(* CODESYS project SingleElevator.project

Project tree, tasks and I/O mapping:
  Device : CODESYS Control Win V3, 3S - Smart Software Solutions GmbH, version 3.5.15.10
    application Application
      libraries: Standard, * (System)
      task MainTask (cyclic, interval 50 ms, priority 1) calls Simulation, GAInstances, Policy
      task VISU_TASK (cyclic, interval 100 ms, priority 31) calls VisuElems.Visu_Prg
      global variables GVL
      visualisation Visualization
      program Simulation [ST]
      function block Motor [SFC]: Closing_active, Closing_exit, Descent_exit, Ascent_active, Ascent_exit, InitFinished_active, Reset_DONEinit_active, Descent_active, Init_active, Ascent_1_active, Descent_1_active, Ready_active, Busy_active, FIN_active, Reset_DONE_active, Ascent_1_exit, CounterUp_active, CounterDown_active, MotStopUp_exit, MotStopDown_exit, Descent_1_exit, Ready_2_active, Busy_2_active, LowSpeed_exit, LowSpeed2_exit, GenCounter_active, ErrDet_active, FaultDeck7_active, Sensor_Fault_active, Error_Floor7_exit, Floor7_active, FloorG_active, AvailableFloor_active, AvailableFloor_exit, FaultDeckG_active, Availablefloor1_active, Availablefloor1_exit
      function block Door [SFC]: Opening_Act_active, Opening_Act_exit, Closing_Act_active, Control_active, Closing_Act_exit, Busy_active, Ready_active, Step1_active, Step1_exit, Init_active, Finished_active, ResetDone_active, Presence_active, Presence_exit, Step3_Closing_Act_active_active, ReOpen_active, ReOpen_exit, Dummy3_exit, ReOpen2_active, ReOpen2_exit
      program Policy [SFC]: Closing_active, Closing_exit, Opening_active, Opening_exit, Motor_Init_exit, Closing_1_active, Closing_1_exit, Upward_active, Upward_exit, Downward_active, Opening_1_active, Opening_1_exit, FloorDetect_active, Motor_Init_active, Downward_exit, ERROR_ARREST_active
      program GAInstances [FBD]
      function block Led [SFC]: GroundFloor_active, Init_active, FirstFloor_active, SecondFloor_active, ThirdFloor_active, FourthFloor_active, FifthFloor_active, SixthFloor_active, SeventhFloor_active, Emergency_active, Ordering_active, Ready_active, Busy_active, Reset_active
  text list GlobalTextList
*)

// Device/Application/GVL
{attribute 'qualified_only'}
VAR_GLOBAL
(* Elevator managing variables*)
	DoorGA_1  	:	Door ;
	MotorGA_1	:	Motor ;
	LedGA_1		:	Led ;

	Open: BOOL;				(* Sensor: the door is fully open*)
	Closed: BOOL;			(* Sensor: the door is fully closed*)
	LimitDown: BOOL;		(* Sensor: lower limit sensor, if TRUE the lift has reached the lower limit*)
	LimitUp: BOOL;			(* Sensor: upper limit sensor, if TRUE the lift has reached the upper limit*)
	DeckSensor: BOOL;		(* Sensor: if TRUE the cab is in proximity of a deck*)
	RampSensor: BOOL;		(* Sensor: if TRUE the cab is in proximity of a ramp*)
	Presence :BOOL; 		(* Sensor: if TRUE something blocks the door photocell*)
	Emergency: BOOL;		(* Input: if TRUE the emergency button has been pressed*)

	Closing: BOOL;			(* Actuator: if TRUE the door starts closing*)
	Opening: BOOL;			(* Actuator: the door starts opening*)
	Motor_on: BOOL;			(* Actuator: if TRUE the lift pulley motor start moving*)
	Up: BOOL;				(* Actuator parameter: if TRUE the lift moves upward, downward otherwise*)
	Vel: BOOL;				(* Actuator parameter: motor speed, if TRUE high speed, low speed otherwise*)


	Current: INT;  			(* Visualization: variable used to storage the current deck*)
    Destination: INT;		(* Visualization: variable used to storage the the destination deck*)
	EmergencyVis: BOOL; 	(* Visualization: if TRUE the emergency light is turned on*)

	InitialDeck: INT := 1;	(* Only for simulation: variable used to define the initial deck*)
	InitCycle: BOOL := FALSE;(* Only for simulation: used to execute the instruction at the first cycle*)
	Height: INT;			(* Only for simulation: elevator height*)
	DeckRest: INT;        	(* Only for simulation: division rest for generating deck sensor*)
	Memory: INT;
	RampRest: INT;			(* Only for simulation: division rest for generating the ramp position*)
	MemoryR: INT;
	Door: INT;				(* Only for simulation: to visualize the closing of the door*)
	Displacement: INT;		(* Only for simulation: lift displacement, dependent on the motor speed*)
	

 (*Inputs: internal panel variables*)
	PG: BOOL;
	P1: BOOL;
	P2: BOOL;
	P3: BOOL;
	P4: BOOL;
	P5: BOOL;
	P6: BOOL;
	P7: BOOL;

(*Visualization: internal panel variables used to turn on the LED*)
	PGVis: BOOL;
	P1Vis: BOOL;
	P2Vis: BOOL;
	P3Vis: BOOL;
	P4Vis: BOOL;
	P5Vis: BOOL;
	P6Vis: BOOL;
	P7Vis: BOOL;

(*Inputs: external panel variables*)
	UpDeckG: BOOL;
	UpDeck1: BOOL;
	UpDeck2: BOOL;
	UpDeck3: BOOL;
	UpDeck4: BOOL;
	UpDeck5: BOOL;
	UpDeck6: BOOL;
	DownDeck7: BOOL;
	DownDeck6: BOOL;
	DownDeck5: BOOL;
	DownDeck4: BOOL;
	DownDeck3: BOOL;
	DownDeck2: BOOL;
	DownDeck1: BOOL;

(*Visualization: external panel variables used to turn on the LED*)
	UpDeckGVis: BOOL;
	UpDeck1Vis: BOOL;
	UpDeck2Vis: BOOL;
	UpDeck3Vis: BOOL;
	UpDeck4Vis: BOOL;
	UpDeck5Vis: BOOL;
	UpDeck6Vis: BOOL;
	DownDeck7Vis: BOOL;
	DownDeck6Vis: BOOL;
	DownDeck5Vis: BOOL;
	DownDeck4Vis: BOOL;
	DownDeck3Vis: BOOL;
	DownDeck2Vis: BOOL;
	DownDeck1Vis: BOOL;

(*Only for simulation: variables used to simulate the fault on deck sensor*)
	SensorG: BOOL;				(* if TRUE the magnetic information for deck G is lost and the deck sensor cannot become TRUE*)
	Sensor1: BOOL;				(* if TRUE the magnetic information for deck 1 is lost and the deck sensor cannot become TRUE*)
	Sensor2: BOOL;
	Sensor3: BOOL;
	Sensor4: BOOL;
	Sensor5: BOOL;
	Sensor6: BOOL;
	Sensor7: BOOL;
	FaultSensorAlarm: BOOL; 	(* Visulaization: if TRUE alerts the user of a deck sensor fault*)

(*Only for simulation: variables used to simulate the fault on ramp sensor*)
	RampGUp: BOOL;
	Ramp1Down: BOOL;
	Ramp1Up:BOOL;
	Ramp2Down: BOOL;
	Ramp2Up:BOOL;
	Ramp3Down: BOOL;
	Ramp3Up:BOOL;
	Ramp4Down: BOOL;
	Ramp4Up:BOOL;
	Ramp5Down: BOOL;
	Ramp5Up:BOOL;
	Ramp6Down: BOOL;
	Ramp6Up:BOOL;
	Ramp7Down: BOOL;
	FaultRampAlarm: BOOL; 		(* Visulaization: if TRUE alerts the user of a ramp sensor fault*)
	SensorGOK: BOOL;
	Sensor1OK: BOOL;
	Sensor2OK: BOOL;
	Sensor6OK: BOOL;
	Sensor3OK: BOOL;
	Sensor4OK: BOOL;
	Sensor5OK: BOOL;
	Sensor7OK: BOOL;
	RampGUpOK: BOOL;
	Ramp1DownOK: BOOL;
	Ramp1UpOK: BOOL;
	Ramp2DownOK: BOOL;
	Ramp2UpOK: BOOL;
	Ramp3DownOK: BOOL;
	Ramp3UpOK: BOOL;
	Ramp4DownOK: BOOL;
	Ramp4UpOK: BOOL;
	Ramp5DownOK: BOOL;
	Ramp5UpOK: BOOL;
	Ramp6DownOK: BOOL;
	Ramp6UpOK: BOOL;
	Ramp7DownOK: BOOL;
	Ramp7UpOK: BOOL;
END_VAR

// Device/Application/Simulation
PROGRAM Simulation
VAR
END_VAR

(* Initial position of the cab inside the hoistway. It is executed only at the first cycle.  *)
IF NOT GVL.InitCycle THEN
			GVL.InitCycle := TRUE ;
			GVL.Height := 20 * GVL.InitialDeck;
		    GVL.Door := 0;
			GVL.Current := GVL.Height / 20;
END_IF;

(* Elevator management, these instructions are executed each cycle time*)

(* Elevator door control. *)
IF GVL.Closing THEN
	GVL.Door := GVL.Door + 1;		(*Closing door management*)
	GVL.Open := FALSE;
END_IF

IF GVL.Door >= 60 THEN						(* Closed door limit*)
	GVL.Closed := TRUE;
END_IF

IF GVL.Opening THEN
	GVL.Door := GVL.Door - 1; 	(* Opening door management*)
	GVL.Closed := FALSE;
END_IF

IF GVL.Door <= 0 THEN							(* Open door limit*)
	GVL.Open := TRUE;
END_IF


(* Maximum and minimum management in the door simulation*)
IF GVL.Door < 0 THEN
	 GVL.Door := 0;
END_IF

IF GVL.Door > 60 THEN
	GVL.Door := 60;
END_IF


(* Control of the cab position inside the hostway. *)
(* Displacement definition for graphic visualization*)
IF GVL.Vel THEN 
	GVL.Displacement := 2;
ELSE 
	GVL.Displacement := 1;
END_IF


(* Height modification relying on direction and speed*)
IF GVL.Motor_on AND GVL.Up THEN
	GVL.Height := GVL.Height + GVL.Displacement;
	GVL.LimitDown := FALSE;
END_IF

IF GVL.Motor_on AND NOT GVL.Up THEN
	GVL.Height := GVL.Height - GVL.Displacement;
	GVL.LimitUp := FALSE;
END_IF


(* Limits for visualization*)
IF GVL.Height < -20 THEN
	GVL.Height := -20;
END_IF

IF GVL.Height > 160 THEN
	GVL.Height := 160;
END_IF

(* Limit sensors management*)
IF GVL.Height <= -10 THEN
	GVL.LimitDown := TRUE;
END_IF

IF GVL.Height >= 150 THEN
	 GVL.LimitUp := TRUE;
END_IF


(*-------------------------------------------------------------------*)
(*  Fault Management (Deck and Ramp Sensors)   *)
(*-------------------------------------------------------------------*)
(* Deck Sensor*)
(* Range of value where the deck sensor is active*)
IF ((GVL.Height >= -1) AND (GVL.Height <= 1)) THEN
	GVL.SensorGOK := TRUE;
ELSE  
	GVL.SensorGOK := FALSE;
END_IF

IF ((GVL.Height >= 20-1) AND (GVL.Height <= 20+1)) THEN
	GVL.Sensor1OK := TRUE;
ELSE  
	GVL.Sensor1OK := FALSE;
END_IF

IF ((GVL.Height >= 40-1) AND (GVL.Height <= 40+1)) THEN
	GVL.Sensor2OK := TRUE;
ELSE  
	GVL.Sensor2OK := FALSE;
END_IF

IF ((GVL.Height >= 60-1) AND (GVL.Height <= 60+1)) THEN
	GVL.Sensor3OK := TRUE;
ELSE  
	GVL.Sensor3OK := FALSE;
END_IF

IF ((GVL.Height >= 80-1) AND (GVL.Height <= 80+1)) THEN
	GVL.Sensor4OK := TRUE;
ELSE  
	GVL.Sensor4OK := FALSE;
END_IF

IF ((GVL.Height >= 100-1) AND (GVL.Height <= 100+1)) THEN
	GVL.Sensor5OK := TRUE;
ELSE   
	GVL.Sensor5OK := FALSE;
END_IF

IF ((GVL.Height >= 120-1) AND (GVL.Height <= 120+1)) THEN
	GVL.Sensor6OK := TRUE;
ELSE  
	GVL.Sensor6OK := FALSE;
END_IF

IF ((GVL.Height >= 140-1) AND (GVL.Height <= 140+1)) THEN
	GVL.Sensor7OK := TRUE;
ELSE  
	GVL.Sensor7OK := FALSE;
END_IF

GVL.DeckSensor := (GVL.SensorGOK AND NOT GVL.SensorG) OR
				    (GVL.Sensor1OK AND NOT GVL.Sensor1) OR
				    (GVL.Sensor2OK AND NOT GVL.Sensor2) OR
				    (GVL.Sensor3OK AND NOT GVL.Sensor3) OR
				    (GVL.Sensor4OK AND NOT GVL.Sensor4) OR
				    (GVL.Sensor5OK AND NOT GVL.Sensor5) OR
				    (GVL.Sensor6OK AND NOT GVL.Sensor6) OR
				    (GVL.Sensor7OK AND NOT GVL.Sensor7);

(* Ramp Sensor*)
(* Range of value where the ramp sensor is active*)
IF ((GVL.Height >= 5-1) AND (GVL.Height <= 5+1)) THEN
	GVL.RampGUpOK := TRUE;
ELSE 
	GVL.RampGUpOK := FALSE;
END_IF

(* Ramp close to deck 1*)
IF ((GVL.Height >= 15-1) AND (GVL.Height <= 15+1)) THEN
	GVL.Ramp1DownOK := TRUE;
ELSE 
	GVL.Ramp1DownOK := FALSE;
END_IF

IF ((GVL.Height >= 25-1) AND (GVL.Height <= 25+1)) THEN
	GVL.Ramp1UpOK := TRUE;
ELSE 
	GVL.Ramp1UpOK := FALSE;
END_IF

(* Ramp close to deck 2*)
IF ((GVL.Height >= 35-1) AND (GVL.Height <= 35+1)) THEN
	GVL.Ramp2DownOK := TRUE;
ELSE 
	GVL.Ramp2DownOK := FALSE;
END_IF

IF ((GVL.Height >= 45-1) AND (GVL.Height <= 45+1)) THEN
	GVL.Ramp2UpOK := TRUE;
ELSE 
	GVL.Ramp2UpOK := FALSE;
END_IF

(*Ramp close to deck  3*)
IF ((GVL.Height >= 55-1) AND (GVL.Height <= 55+1)) THEN
	GVL.Ramp3DownOK := TRUE;
ELSE 
	GVL.Ramp3DownOK := FALSE;
END_IF

IF ((GVL.Height >= 65-1) AND (GVL.Height <= 65+1)) THEN
	GVL.Ramp3UpOK := TRUE;
ELSE 
	GVL.Ramp3UpOK := FALSE;
END_IF

(* Ramp close to deck  4*)
IF ((GVL.Height >= 75-1) AND (GVL.Height <= 75+1)) THEN
	GVL.Ramp4DownOK := TRUE;
ELSE 
	GVL.Ramp4DownOK := FALSE;
END_IF

IF ((GVL.Height >= 85-1) AND (GVL.Height <= 85+1)) THEN
	GVL.Ramp4UpOK := TRUE;
ELSE 
	GVL.Ramp4UpOK:=FALSE;
END_IF

(* Ramp close to deck  5*)
IF ((GVL.Height >= 95-1) AND (GVL.Height <= 95+1)) THEN
	GVL.Ramp5DownOK := TRUE;
ELSE 
	GVL.Ramp5DownOK := FALSE;
END_IF

IF ((GVL.Height >= 105-1) AND (GVL.Height <= 105+1)) THEN
	GVL.Ramp5UpOK := TRUE;
ELSE
	GVL.Ramp5UpOK := FALSE;
END_IF

(* Ramp close to deck  6*)
IF ((GVL.Height >= 115-1) AND (GVL.Height <= 115+1)) THEN
	GVL.Ramp6DownOK := TRUE;
ELSE 
	GVL.Ramp6DownOK := FALSE;
END_IF

IF ((GVL.Height >= 125-1) AND (GVL.Height <= 125+1)) THEN
	GVL.Ramp6UpOK := TRUE;
ELSE 
	GVL.Ramp6UpOK := FALSE;
END_IF

(* Ramp close to deck  7*)
IF ((GVL.Height >= 135-1) AND (GVL.Height <= 135+1)) THEN
	GVL.Ramp7DownOK := TRUE;
ELSE 
	GVL.Ramp7DownOK := FALSE;
END_IF

GVL.RampSensor:=(GVL.RampGUpOK AND NOT GVL.RampGUp) OR 
								(GVL.Ramp1DownOK AND NOT GVL.Ramp1Down ) OR 
								(GVL.Ramp1UpOK AND NOT GVL.Ramp1Up ) OR
								(GVL.Ramp2DownOK AND NOT GVL.Ramp2Down ) OR 
								(GVL.Ramp2UpOK AND NOT GVL.Ramp2Up ) OR
								(GVL.Ramp3DownOK AND NOT GVL.Ramp3Down ) OR
 								(GVL.Ramp3UpOK AND NOT GVL.Ramp3Up ) OR
								(GVL.Ramp4DownOK AND NOT GVL.Ramp4Down ) OR
 								(GVL.Ramp4UpOK AND NOT GVL.Ramp4Up ) OR
								(GVL.Ramp5DownOK AND NOT GVL.Ramp5Down ) OR
 								(GVL.Ramp5UpOK AND NOT GVL.Ramp5Up ) OR
								(GVL.Ramp6DownOK AND NOT GVL.Ramp6Down ) OR
								(GVL.Ramp6UpOK AND NOT GVL.Ramp6Up ) OR
								(GVL.Ramp7DownOK AND NOT GVL.Ramp7Down );

END_PROGRAM

// Device/Application/Door
FUNCTION_BLOCK Door
VAR
	InitDone : BOOL;
END_VAR

VAR_INPUT
	DO_   			: 	BOOL;	
	DOWHAT 			: 	STRING;
	DoorOpen		:	BOOL;
	DoorClosed		:	BOOL;
	Presence		:	BOOL;
END_VAR


VAR_OUTPUT
	DONE 		: 	BOOL;
	State 		: 	STRING;
	OpenDoor	:	BOOL;
	CloseDoor	:	BOOL;
END_VAR

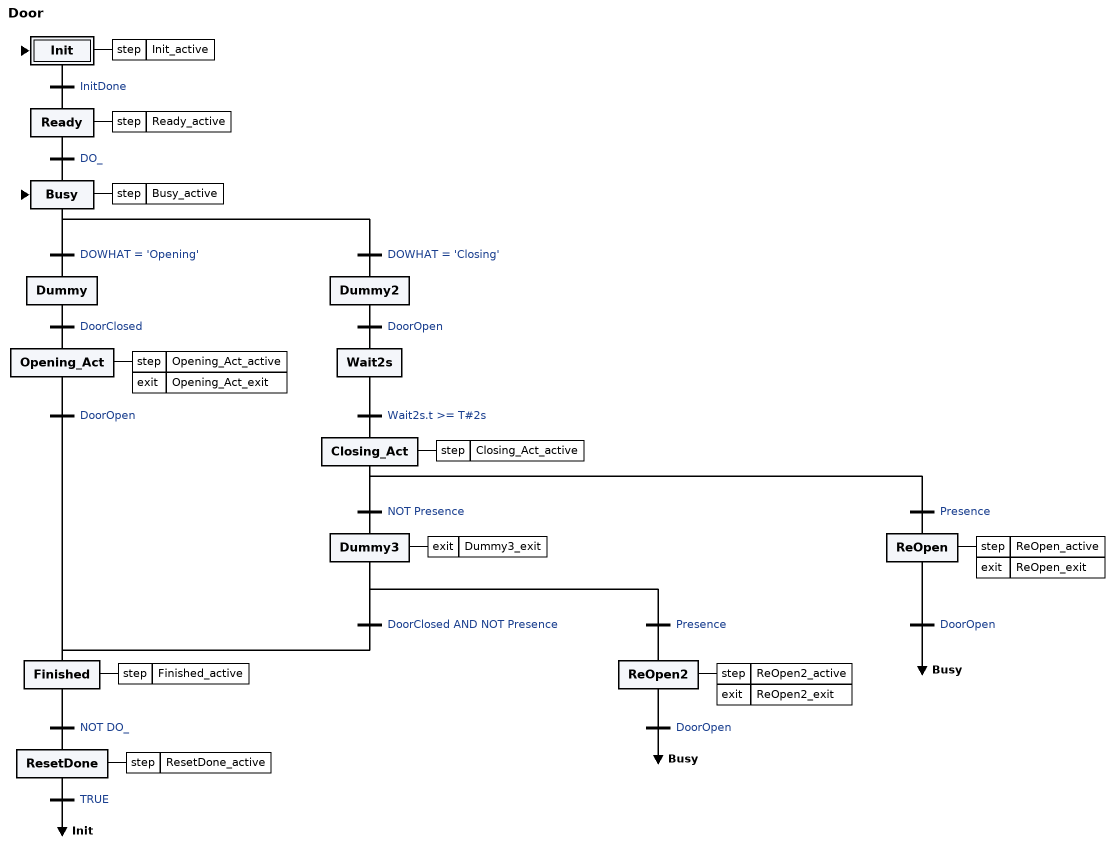
INITIAL_STEP Init:
    Init_active(N);  // step action
END_STEP
TRANSITION FROM Init TO Ready
    := InitDone;
END_TRANSITION
STEP Ready:
    Ready_active(N);  // step action
END_STEP
TRANSITION FROM Ready TO Busy
    := DO_;
END_TRANSITION
STEP Busy:
    Busy_active(N);  // step action
END_STEP
TRANSITION FROM Busy TO Dummy
    := DOWHAT = 'Opening';
END_TRANSITION
STEP Dummy:
END_STEP
TRANSITION FROM Dummy TO Opening_Act
    := DoorClosed;
END_TRANSITION
STEP Opening_Act:
    Opening_Act_active(N);  // step action
    Opening_Act_exit(P0);  // exit action
END_STEP
TRANSITION FROM Opening_Act TO Finished
    := DoorOpen;
END_TRANSITION
TRANSITION FROM Busy TO Dummy2
    := DOWHAT = 'Closing';
END_TRANSITION
STEP Dummy2:
END_STEP
TRANSITION FROM Dummy2 TO Wait2s
    := DoorOpen;
END_TRANSITION
STEP Wait2s:
END_STEP
TRANSITION FROM Wait2s TO Closing_Act
    := Wait2s.t >= T#2s;
END_TRANSITION
STEP Closing_Act:
    Closing_Act_active(N);  // step action
END_STEP
TRANSITION FROM Closing_Act TO Dummy3
    := NOT Presence;
END_TRANSITION
STEP Dummy3:
    Dummy3_exit(P0);  // exit action
END_STEP
TRANSITION FROM Dummy3 TO Finished
    := DoorClosed AND NOT Presence;
END_TRANSITION
TRANSITION FROM Dummy3 TO ReOpen2
    := Presence;
END_TRANSITION
STEP ReOpen2:
    ReOpen2_active(N);  // step action
    ReOpen2_exit(P0);  // exit action
END_STEP
TRANSITION FROM ReOpen2 TO Busy
    := DoorOpen;
END_TRANSITION
TRANSITION FROM Closing_Act TO ReOpen
    := Presence;
END_TRANSITION
STEP ReOpen:
    ReOpen_active(N);  // step action
    ReOpen_exit(P0);  // exit action
END_STEP
TRANSITION FROM ReOpen TO Busy
    := DoorOpen;
END_TRANSITION
STEP Finished:
    Finished_active(N);  // step action
END_STEP
TRANSITION FROM Finished TO ResetDone
    := NOT DO_;
END_TRANSITION
STEP ResetDone:
    ResetDone_active(N);  // step action
END_STEP
TRANSITION FROM ResetDone TO Init
    := TRUE;
END_TRANSITION

ACTION Opening_Act_active:
OpenDoor := TRUE;
END_ACTION

ACTION Opening_Act_exit:
OpenDoor := FALSE;
END_ACTION

ACTION Closing_Act_active:
CloseDoor := TRUE;
END_ACTION

ACTION Control_active:

END_ACTION

ACTION Closing_Act_exit:
GVL.Closing := FALSE;
END_ACTION

ACTION Busy_active:
State := 'Busy';
END_ACTION

ACTION Ready_active:
State := 'Ready';
END_ACTION

ACTION Step1_active:
GVL.Opening := TRUE;
END_ACTION

ACTION Step1_exit:
GVL.Opening := FALSE;
END_ACTION

ACTION Init_active:
State := 'Init';
InitDone := TRUE;
END_ACTION

ACTION Finished_active:
DONE := TRUE;
END_ACTION

ACTION ResetDone_active:
DONE := FALSE;
END_ACTION

ACTION Presence_active:
IF GVL.Presence THEN
	GVL.Closing := FALSE;
	GVL.Opening := TRUE;
END_IF
END_ACTION

ACTION Presence_exit:
GVL.Open := FALSE;
END_ACTION

ACTION Step3_Closing_Act_active_active:

END_ACTION

ACTION ReOpen_active:
CloseDoor := FALSE;
OpenDoor := TRUE;
END_ACTION

ACTION ReOpen_exit:
OpenDoor := FALSE;
END_ACTION

ACTION Dummy3_exit:
CloseDoor := FALSE;
END_ACTION

ACTION ReOpen2_active:
CloseDoor := FALSE;
OpenDoor := TRUE;
END_ACTION

ACTION ReOpen2_exit:
OpenDoor := FALSE;
END_ACTION

END_FUNCTION_BLOCK

// Device/Application/GAInstances
PROGRAM GAInstances
VAR
END_VAR

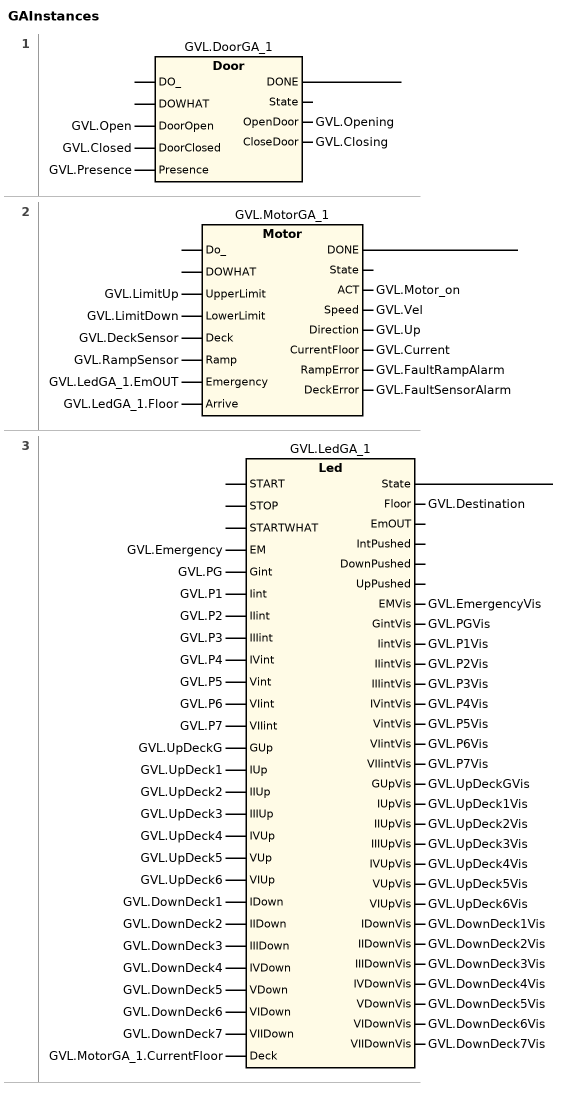
// NETWORK 1
GVL.DoorGA_1(
    DoorOpen := GVL.Open,
    DoorClosed := GVL.Closed,
    Presence := GVL.Presence,
    OpenDoor => GVL.Opening,
    CloseDoor => GVL.Closing); // Door

// NETWORK 2
GVL.MotorGA_1(
    UpperLimit := GVL.LimitUp,
    LowerLimit := GVL.LimitDown,
    Deck := GVL.DeckSensor,
    Ramp := GVL.RampSensor,
    Emergency := GVL.LedGA_1.EmOUT,
    Arrive := GVL.LedGA_1.Floor,
    ACT => GVL.Motor_on,
    Speed => GVL.Vel,
    Direction => GVL.Up,
    CurrentFloor => GVL.Current,
    RampError => GVL.FaultRampAlarm,
    DeckError => GVL.FaultSensorAlarm); // Motor

// NETWORK 3
GVL.LedGA_1(
    EM := GVL.Emergency,
    Gint := GVL.PG,
    Iint := GVL.P1,
    IIint := GVL.P2,
    IIIint := GVL.P3,
    IVint := GVL.P4,
    Vint := GVL.P5,
    VIint := GVL.P6,
    VIIint := GVL.P7,
    GUp := GVL.UpDeckG,
    IUp := GVL.UpDeck1,
    IIUp := GVL.UpDeck2,
    IIIUp := GVL.UpDeck3,
    IVUp := GVL.UpDeck4,
    VUp := GVL.UpDeck5,
    VIUp := GVL.UpDeck6,
    IDown := GVL.DownDeck1,
    IIDown := GVL.DownDeck2,
    IIIDown := GVL.DownDeck3,
    IVDown := GVL.DownDeck4,
    VDown := GVL.DownDeck5,
    VIDown := GVL.DownDeck6,
    VIIDown := GVL.DownDeck7,
    Deck := GVL.MotorGA_1.CurrentFloor,
    Floor => GVL.Destination,
    EMVis => GVL.EmergencyVis,
    GintVis => GVL.PGVis,
    IintVis => GVL.P1Vis,
    IIintVis => GVL.P2Vis,
    IIIintVis => GVL.P3Vis,
    IVintVis => GVL.P4Vis,
    VintVis => GVL.P5Vis,
    VIintVis => GVL.P6Vis,
    VIIintVis => GVL.P7Vis,
    GUpVis => GVL.UpDeckGVis,
    IUpVis => GVL.UpDeck1Vis,
    IIUpVis => GVL.UpDeck2Vis,
    IIIUpVis => GVL.UpDeck3Vis,
    IVUpVis => GVL.UpDeck4Vis,
    VUpVis => GVL.UpDeck5Vis,
    VIUpVis => GVL.UpDeck6Vis,
    IDownVis => GVL.DownDeck1Vis,
    IIDownVis => GVL.DownDeck2Vis,
    IIIDownVis => GVL.DownDeck3Vis,
    IVDownVis => GVL.DownDeck4Vis,
    VDownVis => GVL.DownDeck5Vis,
    VIDownVis => GVL.DownDeck6Vis,
    VIIDownVis => GVL.DownDeck7Vis); // Led

END_PROGRAM

// Device/Application/Motor
FUNCTION_BLOCK Motor


VAR_INPUT
	Do_ 			: 	BOOL;
	DOWHAT 			: 	STRING;
	UpperLimit		:	BOOL;
	LowerLimit		:	BOOL;
	Deck			:	BOOL;
	Ramp			:	BOOL;
	Emergency		: BOOL;
	Arrive			:	INT;
END_VAR

VAR_OUTPUT
	DONE 			: 	BOOL;
	State 			: 	STRING;
	ACT				: 	BOOL;
	Speed			: 	BOOL;
	Direction		: 	BOOL;
	CurrentFloor	:	INT;
	RampError		:   BOOL;
	DeckError		:   BOOL;
END_VAR

VAR
	Decks			: 	ARRAY[0..7] OF BOOL;
	Counter			: 	INT;
	Aux				: 	BOOL;
	InitDone		: 	BOOL; 
	Initia			: 	BOOL;
	CounterDeck 	: 	INT;	
	AuxDeck			: 	BOOL;
	CounterRamp 	: 	INT;
	AuxRamp			:	BOOL;
	RampNumber		:	INT;
	DeckNumber		:	INT;
	Floor 			:	INT;
	n				:	INT;
	AuxRamp1		:	BOOL;
	m				:	INT;
	AuxDeck1		:	BOOL;
	u				: 	INT;
	AuxRamp2		:	BOOL;
	Begin			:	BOOL;
	Upper			:	BOOL;
	Lower			:	BOOL;
	
END_VAR

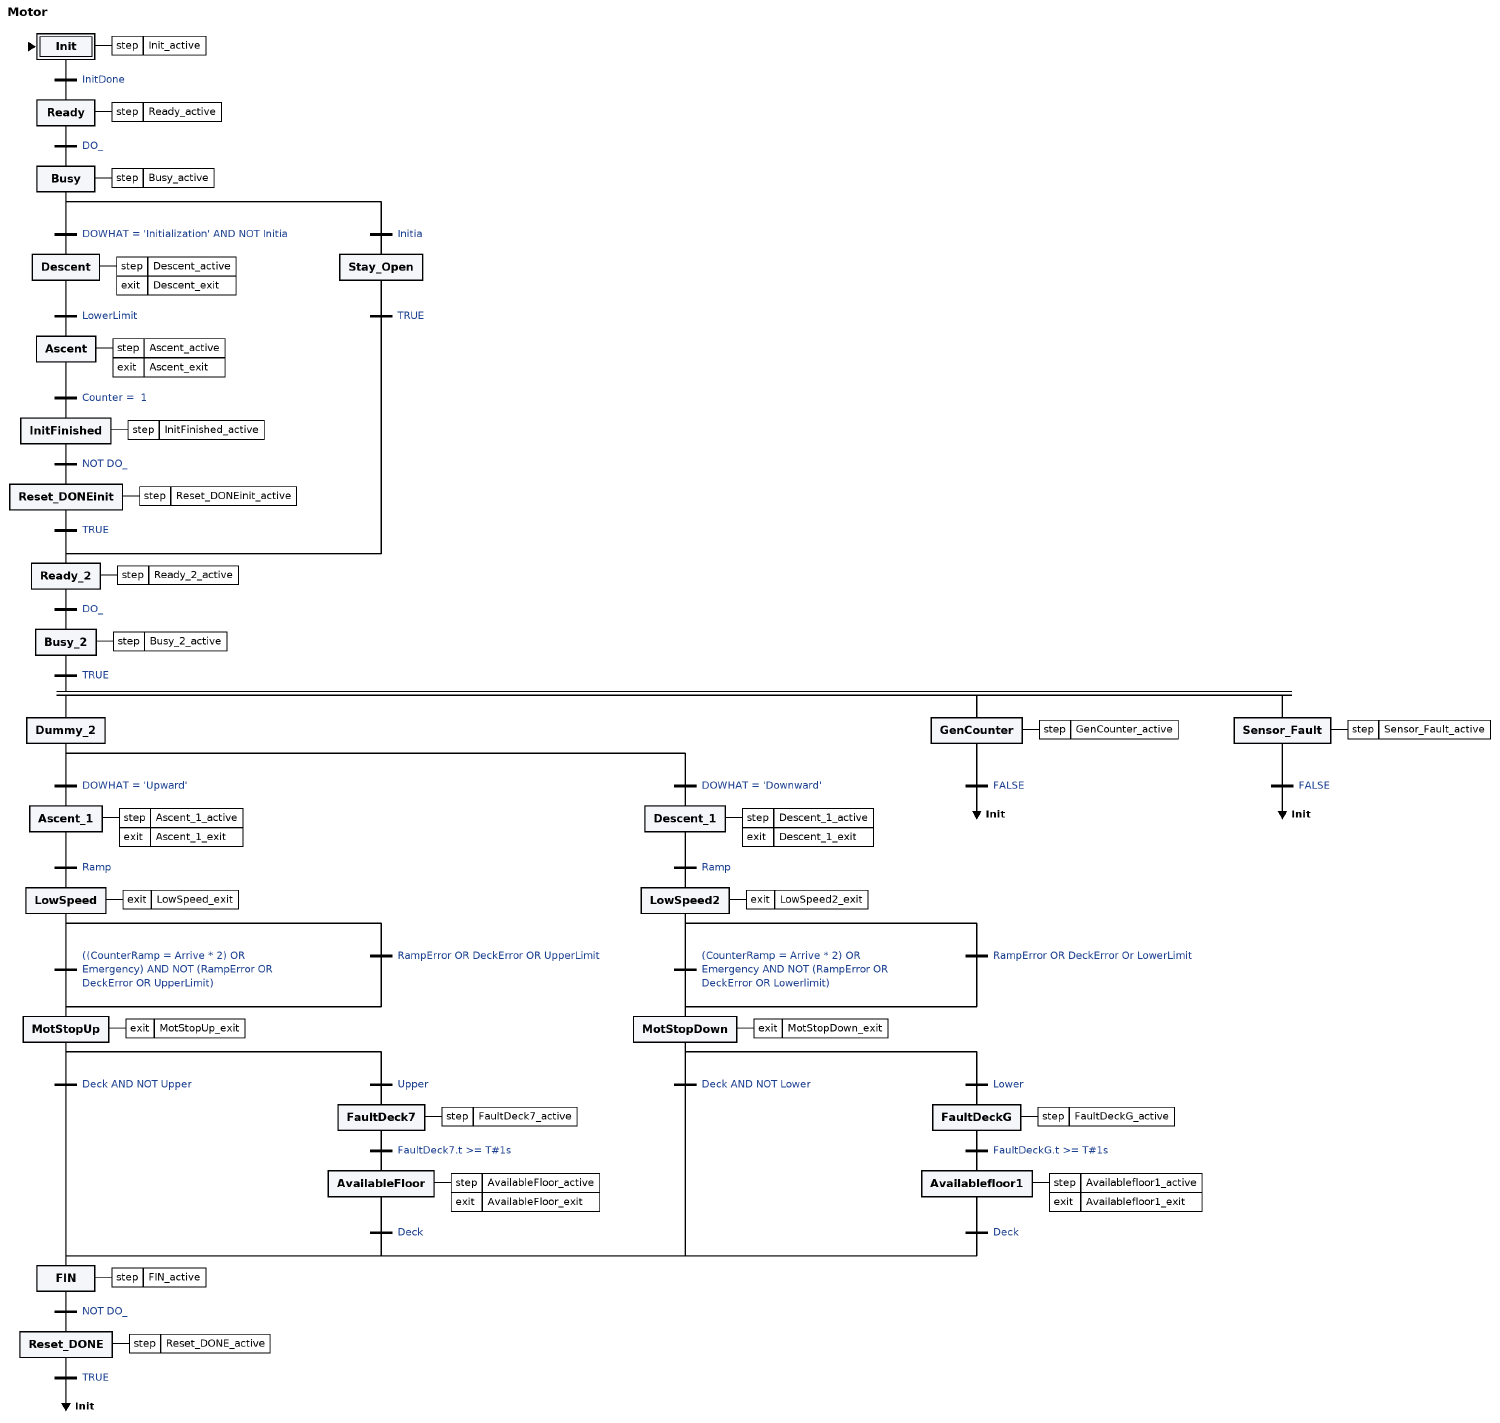
INITIAL_STEP Init:
    Init_active(N);  // step action
END_STEP
TRANSITION FROM Init TO Ready
    := InitDone;
END_TRANSITION
STEP Ready:
    Ready_active(N);  // step action
END_STEP
TRANSITION FROM Ready TO Busy
    := DO_;
END_TRANSITION
STEP Busy:
    Busy_active(N);  // step action
END_STEP
TRANSITION FROM Busy TO Descent
    := DOWHAT = 'Initialization' AND NOT Initia;
END_TRANSITION
STEP Descent:
    Descent_active(N);  // step action
    Descent_exit(P0);  // exit action
END_STEP
TRANSITION FROM Descent TO Ascent
    := LowerLimit;
END_TRANSITION
STEP Ascent:
    Ascent_active(N);  // step action
    Ascent_exit(P0);  // exit action
END_STEP
TRANSITION FROM Ascent TO InitFinished
    := Counter = 1;
END_TRANSITION
STEP InitFinished:
    InitFinished_active(N);  // step action
END_STEP
TRANSITION FROM InitFinished TO Reset_DONEinit
    := NOT DO_;
END_TRANSITION
STEP Reset_DONEinit:
    Reset_DONEinit_active(N);  // step action
END_STEP
TRANSITION FROM Reset_DONEinit TO Ready_2
    := TRUE;
END_TRANSITION
TRANSITION FROM Busy TO Stay_Open
    := Initia;
END_TRANSITION
STEP Stay_Open:
END_STEP
TRANSITION FROM Stay_Open TO Ready_2
    := TRUE;
END_TRANSITION
STEP Ready_2:
    Ready_2_active(N);  // step action
END_STEP
TRANSITION FROM Ready_2 TO Busy_2
    := DO_;
END_TRANSITION
STEP Busy_2:
    Busy_2_active(N);  // step action
END_STEP
TRANSITION FROM Busy_2 TO (Dummy_2, GenCounter, Sensor_Fault)
    := TRUE;
END_TRANSITION
STEP Dummy_2:
END_STEP
STEP GenCounter:
    GenCounter_active(N);  // step action
END_STEP
TRANSITION FROM GenCounter TO Init
    := FALSE;
END_TRANSITION
STEP Sensor_Fault:
    Sensor_Fault_active(N);  // step action
END_STEP
TRANSITION FROM Sensor_Fault TO Init
    := FALSE;
END_TRANSITION
TRANSITION FROM Dummy_2 TO Ascent_1
    := DOWHAT = 'Upward';
END_TRANSITION
STEP Ascent_1:
    Ascent_1_active(N);  // step action
    Ascent_1_exit(P0);  // exit action
END_STEP
TRANSITION FROM Ascent_1 TO LowSpeed
    := Ramp;
END_TRANSITION
STEP LowSpeed:
    LowSpeed_exit(P0);  // exit action
END_STEP
TRANSITION FROM LowSpeed TO MotStopUp
    := ((CounterRamp = Arrive * 2) OR Emergency) AND NOT (RampError OR DeckError OR UpperLimit);
END_TRANSITION
TRANSITION FROM LowSpeed TO MotStopUp
    := RampError OR DeckError OR UpperLimit;
END_TRANSITION
STEP MotStopUp:
    MotStopUp_exit(P0);  // exit action
END_STEP
TRANSITION FROM MotStopUp TO FIN
    := Deck AND NOT Upper;
END_TRANSITION
TRANSITION FROM MotStopUp TO FaultDeck7
    := Upper;
END_TRANSITION
STEP FaultDeck7:
    FaultDeck7_active(N);  // step action
END_STEP
TRANSITION FROM FaultDeck7 TO AvailableFloor
    := FaultDeck7.t >= T#1s;
END_TRANSITION
STEP AvailableFloor:
    AvailableFloor_active(N);  // step action
    AvailableFloor_exit(P0);  // exit action
END_STEP
TRANSITION FROM AvailableFloor TO FIN
    := Deck;
END_TRANSITION
TRANSITION FROM Dummy_2 TO Descent_1
    := DOWHAT = 'Downward';
END_TRANSITION
STEP Descent_1:
    Descent_1_active(N);  // step action
    Descent_1_exit(P0);  // exit action
END_STEP
TRANSITION FROM Descent_1 TO LowSpeed2
    := Ramp;
END_TRANSITION
STEP LowSpeed2:
    LowSpeed2_exit(P0);  // exit action
END_STEP
TRANSITION FROM LowSpeed2 TO MotStopDown
    := (CounterRamp = Arrive * 2) OR Emergency AND NOT (RampError OR DeckError OR Lowerlimit);
END_TRANSITION
TRANSITION FROM LowSpeed2 TO MotStopDown
    := RampError OR DeckError Or LowerLimit;
END_TRANSITION
STEP MotStopDown:
    MotStopDown_exit(P0);  // exit action
END_STEP
TRANSITION FROM MotStopDown TO FIN
    := Deck AND NOT Lower;
END_TRANSITION
TRANSITION FROM MotStopDown TO FaultDeckG
    := Lower;
END_TRANSITION
STEP FaultDeckG:
    FaultDeckG_active(N);  // step action
END_STEP
TRANSITION FROM FaultDeckG TO Availablefloor1
    := FaultDeckG.t >= T#1s;
END_TRANSITION
STEP Availablefloor1:
    Availablefloor1_active(N);  // step action
    Availablefloor1_exit(P0);  // exit action
END_STEP
TRANSITION FROM Availablefloor1 TO FIN
    := Deck;
END_TRANSITION
STEP FIN:
    FIN_active(N);  // step action
END_STEP
TRANSITION FROM FIN TO Reset_DONE
    := NOT DO_;
END_TRANSITION
STEP Reset_DONE:
    Reset_DONE_active(N);  // step action
END_STEP
TRANSITION FROM Reset_DONE TO Init
    := TRUE;
END_TRANSITION

ACTION Closing_active:
GVL.Closing := TRUE;
END_ACTION

ACTION Closing_exit:
GVL.Closing := FALSE;
END_ACTION

ACTION Descent_exit:
ACT := FALSE;
END_ACTION

ACTION Ascent_active:
ACT := TRUE;
Direction := TRUE;

IF Deck AND NOT Aux THEN
	Aux := TRUE;
	Counter := Counter + 1;
END_IF

IF NOT Deck THEN
	Aux := FALSE;
END_IF
END_ACTION

ACTION Ascent_exit:
ACT := FALSE;
END_ACTION

ACTION InitFinished_active:
Initia := TRUE;
DONE := TRUE;
END_ACTION

ACTION Reset_DONEinit_active:
DONE := FALSE;
END_ACTION

ACTION Descent_active:
ACT 		:= TRUE;
Direction 	:= FALSE;
Speed 		:= FALSE;
END_ACTION

ACTION Init_active:
State := 'Init';
InitDone := TRUE;
END_ACTION

ACTION Ascent_1_active:
ACT := TRUE;
Direction := TRUE;
Speed := FALSE;
END_ACTION

ACTION Descent_1_active:
ACT := TRUE;
Direction := FALSE;
Speed := FALSE;
END_ACTION

ACTION Ready_active:
State := 'Ready';
END_ACTION

ACTION Busy_active:
State := 'Busy';
END_ACTION

ACTION FIN_active:
DONE := TRUE;
END_ACTION

ACTION Reset_DONE_active:
DONE := FALSE;
END_ACTION

ACTION Ascent_1_exit:
Speed := TRUE;
END_ACTION

ACTION CounterUp_active:
IF DOWHAT = 'Upward' THEN
	

	IF Deck AND NOT AuxDeck THEN
		AuxDeck := TRUE;
		CounterDeck := CounterDeck + 1;
	END_IF

	IF NOT Deck THEN
		AuxDeck := FALSE;
	END_IF

	IF Ramp AND NOT AuxRamp THEN
		AuxRamp := TRUE;
		CounterRamp := CounterRamp + 1;
	END_IF

	IF NOT Ramp THEN
		AuxRamp := FALSE;
	END_IF

	CurrentFloor := CounterDeck - 1;

END_IF

IF DOWHAT = 'Downward' THEN

	IF Deck AND NOT AuxDeck THEN
		AuxDeck := TRUE;
		CounterDeck := CounterDeck - 1;
	END_IF

	IF NOT Deck THEN
		AuxDeck := FALSE;
	END_IF

	IF Ramp AND NOT AuxRamp THEN
		AuxRamp := TRUE;
		CounterRamp := CounterRamp - 1;
	END_IF

	IF NOT Ramp THEN
		AuxRamp := FALSE;
	END_IF

	CurrentFloor := CounterDeck - 1;

END_IF
END_ACTION

ACTION CounterDown_active:
IF Deck AND NOT AuxDeck THEN
	AuxDeck := TRUE;
	CounterDeck := CounterDeck - 1;
END_IF

IF NOT Deck THEN
	AuxDeck := FALSE;
END_IF

IF Ramp AND NOT AuxRamp THEN
	AuxRamp := TRUE;
	CounterRamp := CounterRamp - 1;
END_IF

IF NOT Ramp THEN
	AuxRamp := FALSE;
END_IF

CurrentFloor := CounterDeck - 1;
END_ACTION

ACTION MotStopUp_exit:
ACT := FALSE;
END_ACTION

ACTION MotStopDown_exit:
ACT := FALSE;
END_ACTION

ACTION Descent_1_exit:
Speed := TRUE;
END_ACTION

ACTION Ready_2_active:
State := 'Ready';
END_ACTION

ACTION Busy_2_active:
State := 'Busy';
END_ACTION

ACTION LowSpeed_exit:
Speed := FALSE;
END_ACTION

ACTION LowSpeed2_exit:
Speed := FALSE;
END_ACTION

ACTION GenCounter_active:
IF DOWHAT = 'Upward' THEN
	

	IF Deck AND NOT AuxDeck THEN
		AuxDeck := TRUE;
		CounterDeck := CounterDeck + 1;
	END_IF

	IF NOT Deck THEN
		AuxDeck := FALSE;
	END_IF

	IF Ramp AND NOT AuxRamp THEN
		AuxRamp := TRUE;
		CounterRamp := CounterRamp + 1;
	END_IF

	IF NOT Ramp THEN
		AuxRamp := FALSE;
	END_IF

	CurrentFloor := CounterDeck - 1;

END_IF

IF DOWHAT = 'Downward' THEN

	IF Deck AND NOT AuxDeck THEN
		AuxDeck := TRUE;
		CounterDeck := CounterDeck - 1;
	END_IF

	IF NOT Deck THEN
		AuxDeck := FALSE;
	END_IF

	IF Ramp AND NOT AuxRamp THEN
		AuxRamp := TRUE;
		CounterRamp := CounterRamp - 1;
	END_IF

	IF NOT Ramp THEN
		AuxRamp := FALSE;
	END_IF

	CurrentFloor := CounterDeck - 1;

END_IF


//IF (RampNumber + 2) <> CounterRamp AND (DeckNumber + 1) <> Counterdeck AND Deck THEN
	//	RampError := TRUE;
//END_IF


// Error detection

//IF (RampNumber + 2) <> CounterRamp AND Deck THEN
//	RampError := TRUE;
//END_IF


(*IF (CurrentFloor + 1) <> CounterDeck THEN
	DeckError := TRUE;

END_IF*)
END_ACTION

ACTION ErrDet_active:
IF (RampNumber + 2) <> CounterRamp THEN
	RampError := TRUE;
END_IF
END_ACTION

ACTION FaultDeck7_active:
ACT := FALSE;
Speed := FALSE;
Direction := FALSE;
END_ACTION

ACTION Sensor_Fault_active:

IF Ramp AND NOT AuxRamp1 THEN
		AuxRamp1 := TRUE;
		n := n + 1; 
END_IF

IF NOT Ramp THEN
		AuxRamp1 := FALSE;
END_IF
	
IF Deck AND NOT AuxDeck1 THEN
	Auxdeck1 := TRUE; 
	m := m + 1;
END_IF

IF NOT Deck THEN 
	Auxdeck1 := FALSE; 
END_IF

IF Deck AND n = 2 THEN
	n := 0;
END_IF

IF NOT Begin AND Ramp THEN
	Begin := TRUE;
	m := 0;
END_IF

IF Deck AND m = 1 AND n = 0 THEN
	m := 0;
END_IF

// IF No Decks are disabled

IF Deck AND m <> 0 AND NOT Upper AND NOT Lower THEN 
	RampError := TRUE;
	n := 0;
END_IF

//IF No Ramps Are Disabled

IF n > 2 THEN
	DeckError := TRUE;
END_IF

// IF arrive = 7 or = G And deck disabled



IF UpperLimit THEN
	Upper := TRUE;
END_IF

IF Upper AND Deck AND  n = 0 THEN
	DeckError := TRUE;
END_IF

IF Upper THEN
	IF Ramp AND NOT AuxRamp2 THEN
		AuxRamp2 := TRUE;
		u := u + 1;
	END_IF

	IF NOT Ramp THEN
		AuxRamp2 := FALSE;
	END_IF
END_IF

IF Upper AND Deck AND  u <> 2 THEN
	RampError := TRUE;
END_IF




IF LowerLimit THEN
	Lower := TRUE;
END_IF

IF Lower AND Deck AND  n = 0 THEN
	DeckError := TRUE;
END_IF

IF Lower THEN
	IF Ramp AND NOT AuxRamp2 THEN
		AuxRamp2 := TRUE;
		u := u + 1;
	END_IF

	IF NOT Ramp THEN
		AuxRamp2 := FALSE;
	END_IF
END_IF

IF Lower AND Deck AND  u <> 2 THEN
	RampError := TRUE;
END_IF
END_ACTION

ACTION Error_Floor7_exit:
ACT := FALSE;
END_ACTION

ACTION Floor7_active:
ACT := TRUE;
Direction := FALSE;
Speed := FALSE;
END_ACTION

ACTION FloorG_active:
ACT := TRUE;
Direction := TRUE;
Speed := FALSE;
END_ACTION

ACTION AvailableFloor_active:
ACT := TRUE;
END_ACTION

ACTION AvailableFloor_exit:
ACT := FALSE;
END_ACTION

ACTION FaultDeckG_active:
ACT := FALSE;
Speed := FALSE;
Direction := TRUE;
END_ACTION

ACTION Availablefloor1_active:
ACT := TRUE;
END_ACTION

ACTION Availablefloor1_exit:
ACT := FALSE;
END_ACTION

END_FUNCTION_BLOCK

// Device/Application/Led
FUNCTION_BLOCK Led

VAR_INPUT
	START		:	BOOL;
	STOP		:	BOOL;
	STARTWHAT	:	STRING;
	EM			:	BOOL;
	Gint		:	BOOL;
	Iint		:	BOOL;
	IIint		:	BOOL;
	IIIint		:	BOOL;
	IVint		:	BOOL;
	Vint		:	BOOL;
	VIint		:	BOOL;
	VIIint		:	BOOL;
	GUp			:	BOOL;
	IUp			:	BOOL;
	IIUp		:	BOOL;
	IIIUp		:	BOOL;
	IVUp		:	BOOL;
	VUp			:	BOOL;
	VIUp		:	BOOL;
	IDown		:	BOOL;
	IIDown		:	BOOL;
	IIIDown		:	BOOL;
	IVDown		:	BOOL;
	VDown		:	BOOL;
	VIDown		:	BOOL;
	VIIDown		:	BOOL;
	Deck		:	INT;
END_VAR

VAR_OUTPUT
	State 			: 	STRING;
	Floor			:	INT;
	EmOUT		:	BOOL;
	IntPushed 		: 	BOOL;
	DownPushed		: 	BOOL;
	UpPushed		:	BOOL;
	EMVis			:	BOOL;
	GintVis			:	BOOL;
	IintVis			:	BOOL;
	IIintVis		:	BOOL;
	IIIintVis		:	BOOL;
	IVintVis		:	BOOL;
	VintVis			:	BOOL;
	VIintVis		:	BOOL;
	VIIintVis		:	BOOL;
	GUpVis			:	BOOL;
	IUpVis			:	BOOL;
	IIUpVis			:	BOOL;
	IIIUpVis		:	BOOL;
	IVUpVis			:	BOOL;
	VUpVis			:	BOOL;
	VIUpVis			:	BOOL;
	IDownVis		:	BOOL;
	IIDownVis		:	BOOL;
	IIIDownVis		:	BOOL;
	IVDownVis		:	BOOL;
	VDownVis		:	BOOL;
	VIDownVis		:	BOOL;
	VIIDownVis		:	BOOL;
END_VAR
VAR
	InitDone	:	BOOL;
	AuxEM		:	BOOL;
	AuxG1		:	BOOL;
	AuxG2		:	BOOL;
	AuxI1		:	BOOL;
	AuxI2		:	BOOL;
	AuxI3		:	BOOL;
	AuxII1		:	BOOL;
	AuxII2		:	BOOL;
	AuxII3		:	BOOL;
	AuxIII1		:	BOOL;
	AuxIII2		:	BOOL;
	AuxIII3		:	BOOL;
	AuxIV1		:	BOOL;
	AuxIV2		:	BOOL;
	AuxIV3		:	BOOL;
	AuxV1		:	BOOL;
	AuxV2		:	BOOL;
	AuxV3		:	BOOL;
	AuxVI1		:	BOOL;
	AuxVI2		:	BOOL;
	AuxVI3		:	BOOL;
	AuxVII1		:	BOOL;
	AuxVII2		:	BOOL;
	AuxVII3		:	BOOL;
	Up_ext 		: 	ARRAY[0..6] OF BOOL; 
	Down_ext	: 	ARRAY[0..7] OF BOOL;
	Intern		: 	ARRAY[0..7] OF BOOL;
	n			:	INT;
	GoDown		:	BOOL;
	
	
END_VAR

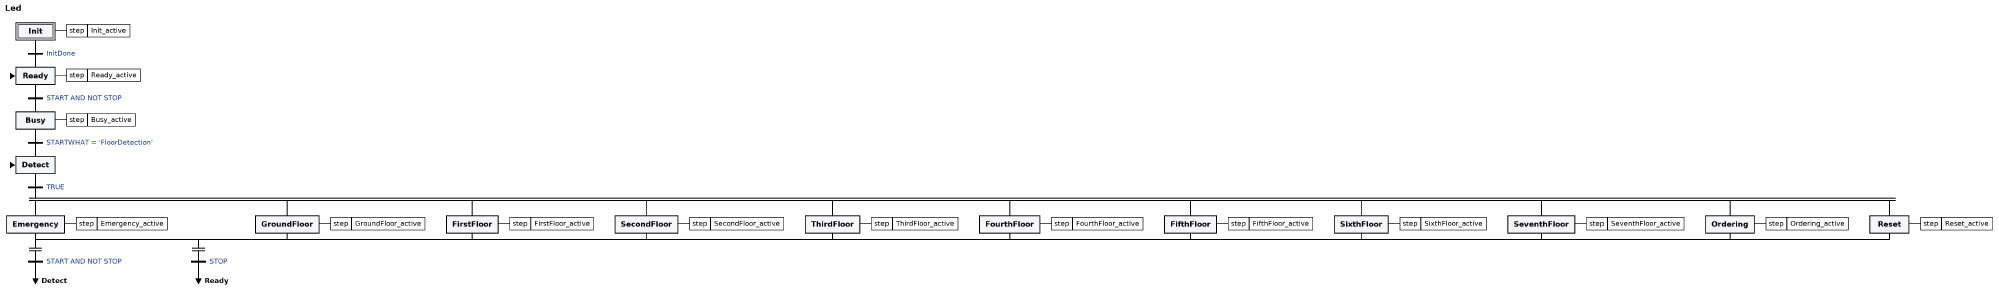
INITIAL_STEP Init:
    Init_active(N);  // step action
END_STEP
TRANSITION FROM Init TO Ready
    := InitDone;
END_TRANSITION
STEP Ready:
    Ready_active(N);  // step action
END_STEP
TRANSITION FROM Ready TO Busy
    := START AND NOT STOP;
END_TRANSITION
STEP Busy:
    Busy_active(N);  // step action
END_STEP
TRANSITION FROM Busy TO Detect
    := STARTWHAT = 'FloorDetection';
END_TRANSITION
STEP Detect:
END_STEP
TRANSITION FROM Detect TO (Emergency, GroundFloor, FirstFloor, SecondFloor, ThirdFloor, FourthFloor, FifthFloor, SixthFloor, SeventhFloor, Ordering, Reset)
    := TRUE;
END_TRANSITION
STEP Emergency:
    Emergency_active(N);  // step action
END_STEP
STEP GroundFloor:
    GroundFloor_active(N);  // step action
END_STEP
STEP FirstFloor:
    FirstFloor_active(N);  // step action
END_STEP
STEP SecondFloor:
    SecondFloor_active(N);  // step action
END_STEP
STEP ThirdFloor:
    ThirdFloor_active(N);  // step action
END_STEP
STEP FourthFloor:
    FourthFloor_active(N);  // step action
END_STEP
STEP FifthFloor:
    FifthFloor_active(N);  // step action
END_STEP
STEP SixthFloor:
    SixthFloor_active(N);  // step action
END_STEP
STEP SeventhFloor:
    SeventhFloor_active(N);  // step action
END_STEP
STEP Ordering:
    Ordering_active(N);  // step action
END_STEP
STEP Reset:
    Reset_active(N);  // step action
END_STEP
TRANSITION FROM (Emergency, GroundFloor, FirstFloor, SecondFloor, ThirdFloor, FourthFloor, FifthFloor, SixthFloor, SeventhFloor, Ordering, Reset) TO Detect
    := START AND NOT STOP;
END_TRANSITION
TRANSITION FROM (Emergency, GroundFloor, FirstFloor, SecondFloor, ThirdFloor, FourthFloor, FifthFloor, SixthFloor, SeventhFloor, Ordering, Reset) TO Ready
    := STOP;
END_TRANSITION

ACTION GroundFloor_active:
IF Gint AND NOT AuxG1 THEN
	AuxG1 := TRUE;
END_IF

IF AuxG1 THEN
	GintVis := TRUE;
	IntPushed := TRUE;
END_IF

IF Floor = 0 AND Deck = 0 THEN 
	GintVis := FALSE;
	AuxG1 := FALSE;
END_IF

IF GUp AND NOT AuxG2 THEN
	AuxG2 := TRUE;
END_IF

IF AuxG2 THEN
	GUpVis := TRUE;
	UpPushed := TRUE;
END_IF

IF Floor = 0 AND Deck = 0 THEN 
	AuxG2 := FALSE;
	IF NOT GoDown THEN
		GUpVis := FALSE;
	END_IF 
END_IF
END_ACTION

ACTION Init_active:
//Remember to change all the buttons with global variable into a simple variable with input variable of the GA the global ones
State := 'Init';
InitDone := TRUE;
END_ACTION

ACTION FirstFloor_active:
IF Iint AND NOT AuxI1 THEN
	AuxI1 := TRUE;
END_IF

IF AuxI1 THEN
	IintVis := TRUE;
	IntPushed := TRUE;
END_IF

IF Floor = 1 AND Deck = 1 THEN 
	IintVis := FALSE;
	AuxI1 := FALSE;
END_IF

IF IUp AND NOT AuxI2 THEN
	AuxI2 := TRUE;
END_IF

IF AuxI2 THEN
	IUpVis := TRUE;
	UpPushed := TRUE;
END_IF

IF Floor = 1 AND Deck = 1 THEN 
	AuxI2 := FALSE;
	IF NOT GoDown THEN
		IUpVis := FALSE;
	END_IF
END_IF

IF IDown AND NOT AuxI3 THEN
	AuxI3 := TRUE;
END_IF

IF AuxI3 THEN
	IDownVis := TRUE;
	DownPushed := TRUE;
END_IF

IF Floor = 1 AND Deck = 1 THEN 
	AuxI3 := FALSE;
	IF GoDown THEN
		IDownVis := FALSE;
	END_IF
END_IF
END_ACTION

ACTION SecondFloor_active:
IF IIint AND NOT AuxII1 THEN
	AuxII1 := TRUE;
END_IF

IF AuxII1 THEN
	IIintVis := TRUE;
	IntPushed := TRUE;
END_IF

IF Floor = 2 AND Deck = 2 THEN 
	IIintVis := FALSE;
	AuxII1 := FALSE;
END_IF

IF IIUp AND NOT AuxII2 THEN
	AuxII2 := TRUE;
END_IF

IF AuxII2 THEN
	IIUpVis := TRUE;
	UpPushed := TRUE;
END_IF

IF Floor = 2 AND Deck = 2 THEN
	AuxII2 := FALSE;
	IF NOT GoDown THEN
		IIUpVis := FALSE;
	END_IF 
END_IF

IF IIDown AND NOT AuxII3 THEN
	AuxII3 := TRUE;
END_IF

IF AuxII3 THEN
	IIDownVis := TRUE;
	DownPushed := TRUE;
END_IF

IF Floor = 2 AND Deck = 2 THEN 
	AuxII3 := FALSE;
	IF GoDown THEN
		IIDownVis := FALSE;
	END_IF
END_IF
END_ACTION

ACTION ThirdFloor_active:
IF IIIint AND NOT AuxIII1 THEN
	AuxIII1 := TRUE;
END_IF

IF AuxIII1 THEN
	IIIintVis := TRUE;
	IntPushed := TRUE;
END_IF

IF Floor = 3 AND Deck = 3 THEN 
	IIIintVis := FALSE;
	AuxIII1 := FALSE;
END_IF

IF IIIUp AND NOT AuxIII2 THEN
	AuxIII2 := TRUE;
END_IF

IF AuxIII2 THEN
	IIIUpVis := TRUE;
	UpPushed := TRUE;
END_IF

IF Floor = 3 AND Deck = 3 THEN 
	AuxIII2 := FALSE;
	IF NOT GoDown THEN
		IIIUpVis := FALSE;
	END_IF 
END_IF

IF IIIDown AND NOT AuxIII3 THEN
	AuxIII3 := TRUE;
END_IF

IF AuxIII3 THEN
	IIIDownVis := TRUE;
	DownPushed := TRUE;
END_IF

IF Floor = 3 AND Deck = 3 THEN 
	AuxIII3 := FALSE;
	IF GoDown THEN
		IIIDownVis := FALSE;
	END_IF
END_IF
END_ACTION

ACTION FourthFloor_active:
IF IVint AND NOT AuxIV1 THEN
	AuxIV1 := TRUE;
END_IF

IF AuxIV1 THEN
	IVintVis := TRUE;
	IntPushed := TRUE;
END_IF

IF Floor = 4 AND Deck = 4 THEN 
	IVintVis := FALSE;
	AuxIV1 := FALSE;
END_IF

IF IVUp AND NOT AuxIV2 THEN
	AuxIV2 := TRUE;
END_IF

IF AuxIV2 THEN
	IVUpVis := TRUE;
	UpPushed := TRUE;
END_IF

IF Floor = 4 AND Deck = 4 THEN 
	AuxIV2 := FALSE;
	IF NOT GoDown THEN
		IVUpVis := FALSE;
	END_IF 
END_IF

IF IVDown AND NOT AuxIV3 THEN
	AuxIV3 := TRUE;
END_IF

IF AuxIV3 THEN
	IVDownVis := TRUE;
	DownPushed := TRUE;
END_IF

IF Floor = 4 AND Deck = 4 THEN
	AuxIV3 := FALSE;
	IF GoDown THEN
		IVDownVis := FALSE;
	END_IF 
END_IF
END_ACTION

ACTION FifthFloor_active:
IF Vint AND NOT AuxV1 THEN
	AuxV1 := TRUE;
END_IF

IF AuxV1 THEN
	VintVis := TRUE;
	IntPushed := TRUE;
END_IF

IF Floor = 5 AND Deck = 5 THEN 
	VintVis := FALSE;
	AuxV1 := FALSE;
END_IF

IF VUp AND NOT AuxV2 THEN
	AuxV2 := TRUE;
END_IF

IF AuxV2 THEN
	VUpVis := TRUE;
	UpPushed := TRUE;
END_IF

IF Floor = 5 AND Deck = 5 THEN 
	AuxV2 := FALSE;
	IF NOT GoDown THEN
		VUpVis := FALSE;
	END_IF 
END_IF

IF VDown AND NOT AuxV3 THEN
	AuxV3 := TRUE;
END_IF

IF AuxV3 THEN
	VDownVis := TRUE;
	DownPushed := TRUE;
END_IF

IF Floor = 5 AND Deck = 5 THEN 
	AuxV3 := FALSE;
	IF GoDown THEN
		VDownVis := FALSE;
	END_IF 
END_IF
END_ACTION

ACTION SixthFloor_active:
IF VIint AND NOT AuxVI1 THEN
	AuxVI1 := TRUE;
END_IF

IF AuxVI1 THEN
	VIintVis := TRUE;
	IntPushed := TRUE;
END_IF

IF Floor = 6 AND Deck = 6 THEN 
	VIintVis := FALSE;
	AuxVI1 := FALSE;
END_IF

IF VIUp AND NOT AuxVI2 THEN
	AuxVI2 := TRUE;
END_IF

IF AuxVI2 THEN
	VIUpVis := TRUE;
	UpPushed := TRUE;
END_IF

IF Floor = 6 AND Deck = 6 THEN 
	AuxVI2 := FALSE;
	IF NOT GoDown THEN
		VIUpVis := FALSE;
	END_IF 
END_IF

IF VIDown AND NOT AuxVI3 THEN
	AuxVI3 := TRUE;
END_IF

IF AuxVI3 THEN
	VIDownVis := TRUE;
	DownPushed := TRUE;
END_IF

IF Floor = 6 AND Deck = 6 THEN 
	AuxVI3 := FALSE;
	IF GoDown THEN
		VIDownVis := FALSE;
	END_IF
END_IF
END_ACTION

ACTION SeventhFloor_active:
IF VIIint AND NOT AuxVII1 THEN
	AuxVII1 := TRUE;
END_IF

IF AuxVII1 THEN
	VIIintVis := TRUE;
	IntPushed := TRUE;
END_IF

IF Floor = 7 AND Deck = 7 THEN 
	VIIintVis := FALSE;
	AuxVII1 := FALSE;
END_IF

IF VIIDown AND NOT AuxVII2 THEN
	AuxVII2 := TRUE;
END_IF

IF AuxVII2 THEN
	VIIDownVis := TRUE;
	DownPushed := TRUE;
END_IF

IF Floor = 7 AND Deck = 7 THEN 
	AuxVII2 := FALSE;
	IF GoDown THEN
		VIIDownVis := FALSE;
	END_IF
END_IF
END_ACTION

ACTION Emergency_active:
IF EM AND NOT AuxEM THEN
	AuxEM := TRUE;
END_IF

IF NOT EM THEN
	AuxEM := FALSE;
END_IF

IF AuxEM THEN
	EmVis := TRUE;
	EmOUT := TRUE;
END_IF

IF NOT AuxEM THEN
	EmVis := FALSE;
	EmOUT := FALSE;
END_IF
END_ACTION

ACTION Ordering_active:

//FILLING ARRAYS

IF Gint THEN
	Intern[0] := TRUE;
END_IF

IF Iint THEN
	Intern[1] := TRUE;
END_IF

IF IIint THEN
	Intern[2] := TRUE;
END_IF

IF IIIint THEN
	Intern[3] := TRUE;
END_IF

IF IVint THEN
	Intern[4] := TRUE;
END_IF

IF Vint THEN
	Intern[5] := TRUE;
END_IF

IF VIint THEN
	Intern[6] := TRUE;
END_IF

IF VIIint THEN
	Intern[7] := TRUE;
END_IF

IF GUp THEN
	Up_ext[0] := TRUE;
END_IF

IF IUp THEN
	Up_ext[1] := TRUE;
END_IF

IF IIUp THEN
	Up_ext[2] := TRUE;
END_IF

IF IIIUp THEN
	Up_ext[3] := TRUE;
END_IF

IF IVUp THEN
	Up_ext[4] := TRUE;
END_IF

IF VUp THEN
	Up_ext[5] := TRUE;
END_IF

IF VIUp THEN
	Up_ext[6] := TRUE;
END_IF

IF IDown THEN
	Down_ext[1] := TRUE;
END_IF

IF IIDown THEN
	Down_ext[2] := TRUE;
END_IF

IF IIIDown THEN
	Down_ext[3] := TRUE;
END_IF

IF IVDown THEN
	Down_ext[4] := TRUE;
END_IF

IF VDown THEN
	Down_ext[5] := TRUE;
END_IF

IF VIDown THEN
	Down_ext[6] := TRUE;
END_IF

IF VIIDown THEN
	Down_ext[7] := TRUE;
END_IF


IF Floor = 0 AND Deck = 0 THEN 
	Intern[0] := FALSE;
	IF NOT GoDown THEN
		Up_ext[0] := FALSE;
	END_IF
END_IF

IF Floor = 1 AND Deck = 1 THEN 
	Intern[1] := FALSE;
	IF NOT GoDown THEN
		Up_ext[1] := FALSE;
	END_IF 
	IF GoDown THEN
		Down_ext[1] := FALSE;
	END_IF 
END_IF

IF Floor = 2 AND Deck = 2 THEN 
	Intern[2] := FALSE;
	IF NOT GoDown THEN
		Up_ext[2] := FALSE;
	END_IF 
	IF GoDown THEN
		Down_ext[2] := FALSE;
	END_IF 
END_IF

IF Floor = 3 AND Deck = 3 THEN 
	Intern[3] := FALSE;
	IF NOT GoDown THEN
		Up_ext[3] := FALSE;
	END_IF
	IF GoDown THEN
		Down_ext[3] := FALSE;
	END_IF	
END_IF

IF Floor = 4 AND Deck = 4 THEN 
	Intern[4] := FALSE;
	IF NOT GoDown THEN
		Up_ext[4] := FALSE;
	END_IF
	IF GoDown THEN
		Down_ext[4] := FALSE;
	END_IF 
END_IF

IF Floor = 5 AND Deck = 5 THEN 
	Intern[5] := FALSE;
	IF NOT GoDown THEN
		Up_ext[5] := FALSE;
	END_IF
	IF GoDown THEN
		Down_ext[5] := FALSE;
	END_IF 
	
END_IF

IF Floor = 6 AND Deck = 6 THEN 
	Intern[6] := FALSE;
	IF NOT GoDown THEN
		Up_ext[6] := FALSE;
	END_IF
	IF GoDown THEN
		Down_ext[6] := FALSE;
	END_IF
	
END_IF

IF Floor = 7 AND Deck = 7 THEN 
	Intern[7] := FALSE;
	IF GoDown THEN
		Down_ext[7] := FALSE;
	END_IF
END_IF


//	CALL DETECTION

	
IF IntPushed OR UpPushed OR DownPushed THEN
	IF NOT GoDown  THEN
		IF Intern[n] OR Up_ext[n] OR (Down_ext[n] AND NOT IntPushed AND NOT UpPushed) THEN
			Floor := n;
			n := Deck;
		ELSE n := n + 1;
		END_IF
		
		IF n > 7 THEN
			n := Deck;
			GoDown := TRUE;
		END_IF
	END_IF

	IF GoDown THEN
		IF Intern[n] OR (Up_ext[n] AND NOT IntPushed AND NOT DownPushed) OR Down_ext[n] THEN
			Floor := n;
			n := Deck;
		ELSE n := n - 1;
		END_IF
			
		IF n < 0 THEN 
			n := Deck;
			GoDown := FALSE;
		END_IF
	END_IF 
END_IF
END_ACTION

ACTION Ready_active:
State := 'Ready';
END_ACTION

ACTION Busy_active:
State := 'Busy';
END_ACTION

ACTION Reset_active:
IF NOT Intern[0] AND NOT Intern[1] AND NOT Intern[2] AND NOT Intern[3] AND NOT Intern[4] AND NOT Intern[5] AND NOT Intern[6] AND NOT Intern[7] THEN
		IntPushed := FALSE;
END_IF

IF NOT Up_ext[0] AND NOT Up_ext[1] AND NOT Up_ext[2] AND NOT Up_ext[3] AND NOT Up_ext[4] AND NOT Up_ext[5] AND NOT Up_ext[6] THEN
	UpPushed := FALSE;
END_IF

IF NOT Down_ext[1] AND NOT Down_ext[2] AND NOT Down_ext[3] AND NOT Down_ext[4] AND NOT Down_ext[5] AND NOT Down_ext[6] AND NOT Down_ext[7] THEN
	DownPushed := FALSE;
END_IF



//IF up > 6 THEN
//	up := 0;
//END_IF

//IF down > 6 THEN
//	down := 0;
//END_IF

//IF in > 7 THEN
//	in := 0;
//END_IF
END_ACTION

END_FUNCTION_BLOCK

// Device/Application/Policy
PROGRAM Policy
VAR
	Synchronization 		:	BOOL;
	OperationOK     		:	BOOL;
	i 						:	INT;
	Call					: 	BOOL;
	Up_ext 					:	ARRAY[0..6] OF BOOL; 
	Down_ext				: 	ARRAY[0..6] OF BOOL;
	Up_int					: 	ARRAY[0..7] OF BOOL;
	Down_int				: 	ARRAY[0..7] OF BOOL;
	InitializationFinished	:	BOOL;
	
END_VAR

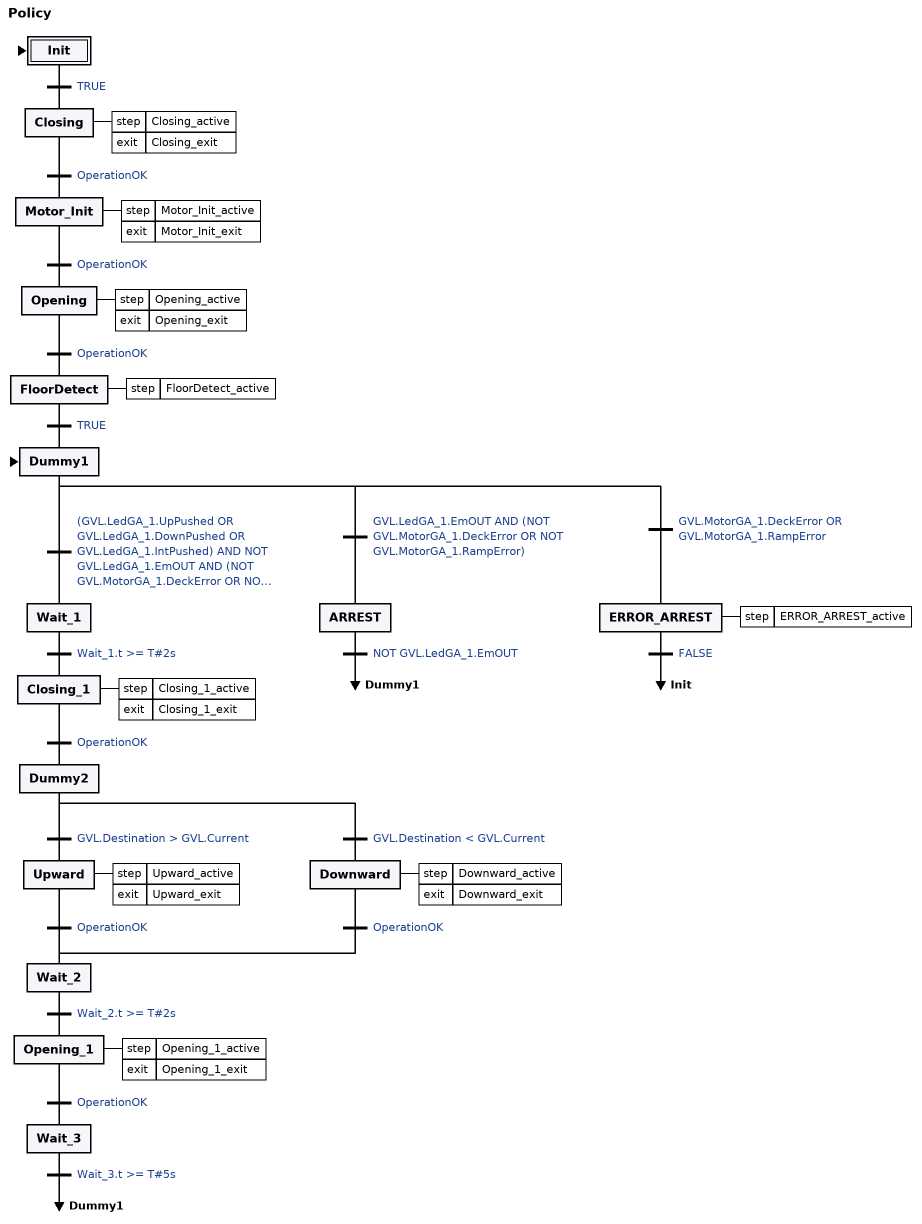
INITIAL_STEP Init:
END_STEP
TRANSITION FROM Init TO Closing
    := TRUE;
END_TRANSITION
STEP Closing:
    Closing_active(N);  // step action
    Closing_exit(P0);  // exit action
END_STEP
TRANSITION FROM Closing TO Motor_Init
    := OperationOK;
END_TRANSITION
STEP Motor_Init:
    Motor_Init_active(N);  // step action
    Motor_Init_exit(P0);  // exit action
END_STEP
TRANSITION FROM Motor_Init TO Opening
    := OperationOK;
END_TRANSITION
STEP Opening:
    Opening_active(N);  // step action
    Opening_exit(P0);  // exit action
END_STEP
TRANSITION FROM Opening TO FloorDetect
    := OperationOK;
END_TRANSITION
STEP FloorDetect:
    FloorDetect_active(N);  // step action
END_STEP
TRANSITION FROM FloorDetect TO Dummy1
    := TRUE;
END_TRANSITION
STEP Dummy1:
END_STEP
TRANSITION FROM Dummy1 TO Wait_1
    := (GVL.LedGA_1.UpPushed OR GVL.LedGA_1.DownPushed OR GVL.LedGA_1.IntPushed) AND NOT GVL.LedGA_1.EmOUT AND (NOT GVL.MotorGA_1.DeckError OR NOT GVL.MotorGA_1.RampError);
END_TRANSITION
TRANSITION FROM Dummy1 TO ARREST
    := GVL.LedGA_1.EmOUT AND (NOT GVL.MotorGA_1.DeckError OR NOT GVL.MotorGA_1.RampError);
END_TRANSITION
STEP ARREST:
END_STEP
TRANSITION FROM ARREST TO Dummy1
    := NOT GVL.LedGA_1.EmOUT;
END_TRANSITION
TRANSITION FROM Dummy1 TO ERROR_ARREST
    := GVL.MotorGA_1.DeckError OR GVL.MotorGA_1.RampError;
END_TRANSITION
STEP ERROR_ARREST:
    ERROR_ARREST_active(N);  // step action
END_STEP
TRANSITION FROM ERROR_ARREST TO Init
    := FALSE;
END_TRANSITION
STEP Wait_1:
END_STEP
TRANSITION FROM Wait_1 TO Closing_1
    := Wait_1.t >= T#2s;
END_TRANSITION
STEP Closing_1:
    Closing_1_active(N);  // step action
    Closing_1_exit(P0);  // exit action
END_STEP
TRANSITION FROM Closing_1 TO Dummy2
    := OperationOK;
END_TRANSITION
STEP Dummy2:
END_STEP
TRANSITION FROM Dummy2 TO Upward
    := GVL.Destination > GVL.Current;
END_TRANSITION
STEP Upward:
    Upward_active(N);  // step action
    Upward_exit(P0);  // exit action
END_STEP
TRANSITION FROM Upward TO Wait_2
    := OperationOK;
END_TRANSITION
TRANSITION FROM Dummy2 TO Downward
    := GVL.Destination < GVL.Current;
END_TRANSITION
STEP Downward:
    Downward_active(N);  // step action
    Downward_exit(P0);  // exit action
END_STEP
TRANSITION FROM Downward TO Wait_2
    := OperationOK;
END_TRANSITION
STEP Wait_2:
END_STEP
TRANSITION FROM Wait_2 TO Opening_1
    := Wait_2.t >= T#2s;
END_TRANSITION
STEP Opening_1:
    Opening_1_active(N);  // step action
    Opening_1_exit(P0);  // exit action
END_STEP
TRANSITION FROM Opening_1 TO Wait_3
    := OperationOK;
END_TRANSITION
STEP Wait_3:
END_STEP
TRANSITION FROM Wait_3 TO Dummy1
    := Wait_3.t >= T#5s;
END_TRANSITION

ACTION Closing_active:
IF GVL.DoorGA_1.State = 'Ready' THEN
	GVL.DoorGA_1.DO_ := TRUE;
	GVL.DoorGA_1.DOWHAT := 'Closing';
END_IF


IF (GVL.DoorGA_1.State = 'Busy') AND (GVL.DoorGA_1.DONE = TRUE) THEN
	GVL.DoorGA_1.DO_ := FALSE;
	Synchronization := TRUE;
END_IF


OperationOK := Synchronization AND NOT GVL.DoorGA_1.DONE;
END_ACTION

ACTION Closing_exit:
Synchronization := FALSE;
OperationOK := FALSE;
END_ACTION

ACTION Opening_active:
IF GVL.DoorGA_1.State = 'Ready' THEN
	GVL.DoorGA_1.DO_ := TRUE;
	GVL.DoorGA_1.DOWHAT := 'Opening';
END_IF


IF (GVL.DoorGA_1.State = 'Busy') AND (GVL.DoorGA_1.DONE = TRUE) THEN
	GVL.DoorGA_1.DO_ := FALSE;
	Synchronization := TRUE;
END_IF


OperationOK := Synchronization AND NOT GVL.DoorGA_1.DONE;
END_ACTION

ACTION Opening_exit:
Synchronization := FALSE;
OperationOK := FALSE;
END_ACTION

ACTION Motor_Init_exit:
Synchronization := FALSE;
OperationOK := FALSE;
END_ACTION

ACTION Closing_1_active:
IF GVL.DoorGA_1.State = 'Ready' THEN
	GVL.DoorGA_1.DO_ := TRUE;
	GVL.DoorGA_1.DOWHAT := 'Closing';
END_IF


IF (GVL.DoorGA_1.State = 'Busy') AND (GVL.DoorGA_1.DONE = TRUE) THEN
	GVL.DoorGA_1.DO_ := FALSE;
	Synchronization := TRUE;
END_IF


OperationOK := Synchronization AND NOT GVL.DoorGA_1.DONE;
END_ACTION

ACTION Closing_1_exit:
Synchronization := FALSE;
OperationOK := FALSE;
END_ACTION

ACTION Upward_active:
IF GVL.MotorGA_1.State = 'Ready' THEN
	GVL.MotorGA_1.DO_ := TRUE;
	GVL.MotorGA_1.DOWHAT := 'Upward';
END_IF


IF (GVL.MotorGA_1.State = 'Busy') AND (GVL.MotorGA_1.DONE = TRUE) THEN
	GVL.MotorGA_1.DO_ := FALSE;
	Synchronization := TRUE;
END_IF


OperationOK := Synchronization AND NOT GVL.MotorGA_1.DONE;
END_ACTION

ACTION Upward_exit:
Synchronization := FALSE;
OperationOK := FALSE;
END_ACTION

ACTION Downward_active:
IF GVL.MotorGA_1.State = 'Ready' THEN
	GVL.MotorGA_1.DO_ := TRUE;
	GVL.MotorGA_1.DOWHAT := 'Downward';
END_IF


IF (GVL.MotorGA_1.State = 'Busy') AND (GVL.MotorGA_1.DONE = TRUE) THEN
	GVL.MotorGA_1.DO_ := FALSE;
	Synchronization := TRUE;
END_IF


OperationOK := Synchronization AND NOT GVL.MotorGA_1.DONE;
END_ACTION

ACTION Opening_1_active:
IF GVL.DoorGA_1.State = 'Ready' THEN
	GVL.DoorGA_1.DO_ := TRUE;
	GVL.DoorGA_1.DOWHAT := 'Opening';
END_IF


IF (GVL.DoorGA_1.State = 'Busy') AND (GVL.DoorGA_1.DONE = TRUE) THEN
	GVL.DoorGA_1.DO_ := FALSE;
	Synchronization := TRUE;
END_IF


OperationOK := Synchronization AND NOT GVL.DoorGA_1.DONE;
END_ACTION

ACTION Opening_1_exit:
Synchronization := FALSE;
OperationOK := FALSE;
END_ACTION

ACTION FloorDetect_active:
IF GVL.LedGA_1.State = 'Ready' THEN
	GVL.LedGA_1.START := TRUE;
	GVL.LedGA_1.STOP := FALSE;
	GVL.LedGA_1.STARTWHAT := 'FloorDetection';
END_IF
END_ACTION

ACTION Motor_Init_active:
IF GVL.MotorGA_1.State = 'Ready' THEN
	GVL.MotorGA_1.DO_ := TRUE;
	GVL.MotorGA_1.DOWHAT := 'Initialization';
END_IF


IF (GVL.MotorGA_1.State = 'Busy') AND (GVL.MotorGA_1.DONE = TRUE) THEN
	GVL.MotorGA_1.DO_ := FALSE;
	Synchronization := TRUE;
END_IF


OperationOK := Synchronization AND NOT GVL.MotorGA_1.DONE;
END_ACTION

ACTION Downward_exit:
Synchronization := FALSE;
OperationOK := FALSE;
END_ACTION

ACTION ERROR_ARREST_active:
GVL.LedGA_1.START := FALSE;
GVL.LedGA_1.STOP := TRUE;
END_ACTION

END_PROGRAM

// Device/Application/Visualization
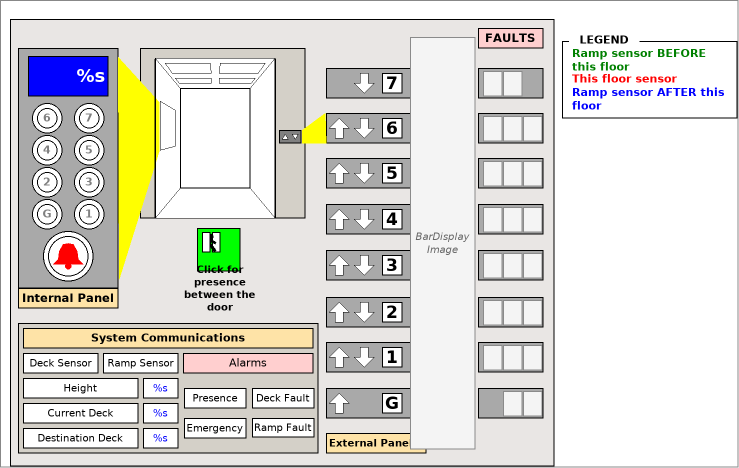
VISUALIZATION Visualization  // 739x468
    Rectangle (10,19 544x447)
    Rectangle (197,228 43x43), colour toggle: GVL.Presence
    Rectangle (18,323 300x130)
    Rectangle (326,433 100x20), "External Panels"
    Rectangle (326,342 100x30)
    Rectangle (382,347 20x20), "1"
    Polygon (354,357) (360,357) (360,347) (368,347) (368,357) (374,357) (364,367), colour toggle: GVL.DownDeck1Vis
        tap GVL.DownDeck1
    Polygon (329,357) (335,357) (335,367) (343,367) (343,357) (349,357) (339,347), colour toggle: GVL.UpDeck1Vis
        tap GVL.UpDeck1
    Rectangle (326,297 100x30)
    Rectangle (382,302 20x20), "2"
    Polygon (354,312) (360,312) (360,302) (368,302) (368,312) (374,312) (364,322), colour toggle: GVL.DownDeck2Vis
        tap GVL.DownDeck2
    Polygon (329,312) (335,312) (335,322) (343,322) (343,312) (349,312) (339,302), colour toggle: GVL.UpDeck2Vis
        tap GVL.UpDeck2
    Rectangle (326,250 100x30)
    Rectangle (382,255 20x20), "3"
    Polygon (354,265) (360,265) (360,255) (368,255) (368,265) (374,265) (364,275), colour toggle: GVL.DownDeck3Vis
        tap GVL.DownDeck3
    Polygon (329,265) (335,265) (335,275) (343,275) (343,265) (349,265) (339,255), colour toggle: GVL.UpDeck3Vis
        tap GVL.UpDeck3
    Rectangle (326,204 100x30)
    Rectangle (382,209 20x20), "4"
    Polygon (354,219) (360,219) (360,209) (368,209) (368,219) (374,219) (364,229), colour toggle: GVL.DownDeck4Vis
        tap GVL.DownDeck4
    Polygon (329,219) (335,219) (335,229) (343,229) (343,219) (349,219) (339,209), colour toggle: GVL.UpDeck4Vis
        tap GVL.UpDeck4
    Rectangle (326,158 100x30)
    Rectangle (382,163 20x20), "5"
    Polygon (354,173) (360,173) (360,163) (368,163) (368,173) (374,173) (364,183), colour toggle: GVL.DownDeck5Vis
        tap GVL.DownDeck5
    Polygon (329,173) (335,173) (335,183) (343,183) (343,173) (349,173) (339,163), colour toggle: GVL.UpDeck5Vis
        tap GVL.UpDeck5
    Rectangle (326,113 100x30)
    Rectangle (382,118 20x20), "6"
    Polygon (354,128) (360,128) (360,118) (368,118) (368,128) (374,128) (364,138), colour toggle: GVL.DownDeck6Vis
        tap GVL.DownDeck6
    Polygon (329,128) (335,128) (335,138) (343,138) (343,128) (349,128) (339,118), colour toggle: GVL.UpDeck6Vis
        tap GVL.UpDeck6
    Rectangle (326,68 100x30)
    Rectangle (382,73 20x20), "7"
    Polygon (354,83) (360,83) (360,73) (368,73) (368,83) (374,83) (364,93), colour toggle: GVL.DownDeck7Vis
        tap GVL.DownDeck7
    Rectangle (326,388 100x30)
    Rectangle (382,393 20x20), "G"
    Polygon (329,403) (335,403) (335,413) (343,413) (343,403) (349,403) (339,393), colour toggle: GVL.UpDeckGVis
        tap GVL.UpDeckG
    RoundedRectangle (18,48 100x240)
    Rectangle (18,288 100x20), "Internal Panel"
    Ellipse (74,199 30x30), colour toggle: GVL.P1Vis
    Ellipse (79,204 20x20), "1"
        tap GVL.P1
    Ellipse (32,199 30x30), colour toggle: GVL.PGVis
    Ellipse (37,204 20x20), "G"
        tap GVL.PG
    Ellipse (74,167 30x30), colour toggle: GVL.P3Vis
    Ellipse (79,172 20x20), "3"
        tap GVL.P3
    Ellipse (32,167 30x30), colour toggle: GVL.P2Vis
    Ellipse (37,172 20x20), "2"
        tap GVL.P2
    Ellipse (74,135 30x30), colour toggle: GVL.P5Vis
    Ellipse (79,140 20x20), "5"
        tap GVL.P5
    Ellipse (32,135 30x30), colour toggle: GVL.P4Vis
    Ellipse (37,140 20x20), "4"
        tap GVL.P4
    Ellipse (74,103 30x30), colour toggle: GVL.P7Vis
    Ellipse (79,108 20x20), "7"
        tap GVL.P7
    Ellipse (32,103 30x30), colour toggle: GVL.P6Vis
    Ellipse (37,108 20x20), "6"
        tap GVL.P6
    Rectangle (28,56 80x40), "%s", text variable: GVL.Destination
    Ellipse (43,231 50x50), tooltip "EMERGENCY", colour toggle: GVL.Emergency
    Group (48,236 40x40)
        toggle GVL.Emergency
        Ellipse (0,0 40x40), tooltip "EMERGENCY"
        Polygon (5,28) (10,23) (11,15) (15,8) (20,7) (25,8) (29,15) (30,23) (35,28)
        Ellipse (17,27 6x6)
    Polygon (35,72) (45,62) (55,72), colour toggle: GVL.Motor_on AND GVL.Up
    Polygon (35,80) (45,90) (55,80), colour toggle: GVL.Motor_on AND NOT GVL.Up
    Group (140,48 165x170)
        Rectangle (0,0 165x170)
        Rectangle (15,10 120x160)
        Polygon (40,40) (15,10) (135,10) (110,40)
        Rectangle (40,40 70x100)
        Polygon (15,170) (40,140) (110,140) (135,170)
        Polygon (20,102) (20,53) (35,62) (35,98)
        Polygon (79,35) (79,30) (115,30) (111,35)
        Polygon (39,35) (35,30) (71,30) (71,35)
        Polygon (32,25) (25,15) (70,15) (71,25)
        Polygon (79,25) (80,15) (125,15) (118,25)
        Group (139,82 22x13)
            Rectangle (0,0 22x13)
            Polygon (3,9) (6,4) (9,9)
            Polygon (13,4) (16,9) (19,4)
    BarDisplayImage (410,37 65x412), value: GVL.Height, style: BarDisplayImage-Gray, scale format: %.0f, scale -20..160
        p3451962224: VisuNativeControl.IP_Offline.Browser
    Rectangle (478,68 65x30)
    Rectangle (478,342 65x30)
    Rectangle (478,297 65x30)
    Rectangle (478,250 65x30)
    Rectangle (478,204 65x30)
    Rectangle (478,158 65x30)
    Rectangle (478,113 65x30)
    Rectangle (478,388 65x30)
    RockerSwitch (483,345 19x25), variable: GVL.Ramp1Down, behaviour: TOGGLE, style: Switch-RockerSwitch-Green
    RockerSwitch (503,345 19x25), variable: GVL.Sensor1, behaviour: TOGGLE, style: Switch-RockerSwitch-Red
    RockerSwitch (523,345 19x25), variable: GVL.Ramp1Up, behaviour: TOGGLE, style: Switch-RockerSwitch-Blue
    RockerSwitch (483,300 19x25), variable: GVL.Ramp2Down, behaviour: TOGGLE, style: Switch-RockerSwitch-Green
    RockerSwitch (503,300 19x25), variable: GVL.Sensor2, behaviour: TOGGLE, style: Switch-RockerSwitch-Red
    RockerSwitch (523,300 19x25), variable: GVL.Ramp2Up, behaviour: TOGGLE, style: Switch-RockerSwitch-Blue
    RockerSwitch (483,253 19x25), variable: GVL.Ramp3Down, behaviour: TOGGLE, style: Switch-RockerSwitch-Green
    RockerSwitch (503,253 19x25), variable: GVL.Sensor3, behaviour: TOGGLE, style: Switch-RockerSwitch-Red
    RockerSwitch (523,253 19x25), variable: GVL.Ramp3Up, behaviour: TOGGLE, style: Switch-RockerSwitch-Blue
    RockerSwitch (483,207 19x25), variable: GVL.Ramp4Down, behaviour: TOGGLE, style: Switch-RockerSwitch-Green
    RockerSwitch (503,207 19x25), variable: GVL.Sensor4, behaviour: TOGGLE, style: Switch-RockerSwitch-Red
    RockerSwitch (523,207 19x25), variable: GVL.Ramp4Up, behaviour: TOGGLE, style: Switch-RockerSwitch-Blue
    RockerSwitch (483,161 19x25), variable: GVL.Ramp5Down, behaviour: TOGGLE, style: Switch-RockerSwitch-Green
    RockerSwitch (503,161 19x25), variable: GVL.Sensor5, behaviour: TOGGLE, style: Switch-RockerSwitch-Red
    RockerSwitch (523,161 19x25), variable: GVL.Ramp5Up, behaviour: TOGGLE, style: Switch-RockerSwitch-Blue
    RockerSwitch (483,116 19x25), variable: GVL.Ramp6Down, behaviour: TOGGLE, style: Switch-RockerSwitch-Green
    RockerSwitch (503,116 19x25), variable: GVL.Sensor6, behaviour: TOGGLE, style: Switch-RockerSwitch-Red
    RockerSwitch (523,116 19x25), variable: GVL.Ramp6Up, behaviour: TOGGLE, style: Switch-RockerSwitch-Blue
    RockerSwitch (483,71 19x25), variable: GVL.Ramp7Down, behaviour: TOGGLE, style: Switch-RockerSwitch-Green
    RockerSwitch (503,71 19x25), variable: GVL.Sensor7, behaviour: TOGGLE, style: Switch-RockerSwitch-Red
    RockerSwitch (503,391 19x25), variable: GVL.SensorG, behaviour: TOGGLE, style: Switch-RockerSwitch-Red
    RockerSwitch (523,391 19x25), variable: GVL.RampGUp, behaviour: TOGGLE, style: Switch-RockerSwitch-Blue
    Rectangle (478,28 65x20), "FAULTS"
    Polygon (302,130) (325,113) (326,143) (302,143), invisible if: (GVL.Closing OR GVL.Opening) OR GVL.Closed
    Polygon (118,57) (159,102) (159,151) (119,279), invisible if: (GVL.Closing OR GVL.Opening) OR GVL.Closed
    Rectangle (155,58 0x160)
        p3528305787: GVL.Door
    Rectangle (275,58 0x160)
        p3528305787: -GVL.Door
    Rectangle (23,328 290x20), "System Communications"
    Rectangle (183,353 130x20), "Alarms"
    Rectangle (23,353 75x20), "Deck Sensor", colour toggle: GVL.DeckSensor
    Rectangle (143,378 35x20), "%s", text variable: GVL.Height
    Rectangle (184,388 62x20), "Presence", colour toggle: GVL.Presence
    Rectangle (103,353 75x20), "Ramp Sensor", colour toggle: GVL.RampSensor
    Rectangle (143,403 35x20), "%s", text variable: GVL.Current
    Rectangle (143,428 35x20), "%s", text variable: GVL.Destination
    Rectangle (252,388 62x20), "Deck Fault", colour toggle: GVL.FaultSensorAlarm
    Rectangle (184,418 62x20), "Emergency", colour toggle: GVL.EmergencyVis
    Rectangle (252,418 62x19), "Ramp Fault", colour toggle: GVL.FaultRampAlarm
    Rectangle (23,378 115x20), "Height"
    Rectangle (23,403 115x20), "Current Deck"
    Rectangle (23,428 115x20), "Destination Deck"
    Group (562,25 175x93)
        Rectangle (0,16 175x77)
        Rectangle (7,39 160x30), "This floor sensor"
        Rectangle (7,59 160x30), "Ramp sensor AFTER this floor"
        Rectangle (7,0 70x30), "LEGEND"
        Rectangle (7,20 160x30), "Ramp sensor BEFORE this floor"
    Group (202,232 33x34)
        toggle GVL.Presence
        Rectangle (10,0 8x20)
        Polygon (5,10) (12,20) (14,18) (5,6)
        Ellipse (6,2 5x5)
        Polygon (4,8) (13,12) (14,10) (4,4)
        Rectangle (0,0 8x20)
    Rectangle (169,273 102x31), "Click for presence between the door"
END_VISUALIZATION
